{attribute 'linkalways'} 
{attribute 'no_explicit_call' := 'This FB is a CLASS and must be accessed using methods or properties'}
{attribute 'enable_dynamic_creation'}
FUNCTION_BLOCK Node_F_VN_DetectBlobsExp EXTENDS VisionNode
VAR
    ipSrcImage : _ITcVnImage;
    ipBlobContours : _ITcVnContainer;
    stParams : _TcVnParamsBlobDetection;
    aOffset : _TcVnPoint;
    hrPrev : _HRESULT(S_OK);
	hresult : _HRESULT(S_OK);
END_VAR

METHOD PUBLIC  Clone : I_Node
VAR
	pNode : POINTER TO Node_F_VN_DetectBlobsExp;
END_VAR
pNode := __NEW(Node_F_VN_DetectBlobsExp);
Clone := pNode^;
END_METHOD

METHOD FB_init : BOOL
VAR_INPUT
	bInitRetains : BOOL; // if TRUE, the retain variables are initialized (warm start / cold start)
	bInCopyCode : BOOL;  // if TRUE, the instance afterwards gets moved into the copy code (online change)
END_VAR
AddInput('ipSrcImage', ipSrcImage);
AddInput('stParams', stParams);
AddInput('aOffset', aOffset);
AddInput('hrPrev', hrPrev);
AddOutput('ipBlobContours', ipBlobContours);
AddOutput('hresult', hresult);
END_METHOD

METHOD PROTECTED OnExecute
hresult.Value := F_VN_DetectBlobsExp(
	ipSrcImage := ipSrcImage.Value,
    ipBlobContours := ipBlobContours.Value,
    stParams := stParams.Value,
    aOffset := aOffset.Value,
	hrPrev:= hrPrev.Value);
END_METHOD

METHOD PUBLIC PreExecutionCheck
VAR_INPUT
	Check : I_PreExecutionChecks;
END_VAR
Check.IsTrue(ipSrcImage.IsValid, 'ipSrcImage must contain an image');
Check.IsTrue((ipSrcImage.IsPixelDepth(8) OR ipSrcImage.IsPixelDepth(32)), 'ipSrcImage must be 8 or 32 bit pixel depth');
Check.IsTrue((ipSrcImage.HasChannelCount(1) OR ipSrcImage.HasChannelCount(3)), 'ipSrcImage must contain 1 or 3 channels');
Check.IsTrue(stParams.Value.fMaxThreshold >= stParams.Value.fMinThreshold, 'fMaxThreshold must be greater than or equal to fMinThreshold');
END_METHOD

END_FUNCTION_BLOCK

(* stored: Version 1.1.0.1, ProductVersion 3.1.4026.18
   POU Node_F_VN_DetectBlobsExp: Id {a7966657-125c-0d2b-32fa-81ffe10221c8}, SpecialFunc None
   Folder Constructor: Id {bbc10436-0102-05b7-2a51-3c32a270b36e}
   Method Clone: Id {25bd43b8-17ef-0404-3b99-a3d69c5d11e2}
   Method FB_init: Id {25aaaa77-b7d6-07c3-10e2-a0f8986286a8}
   Method OnExecute: Id {c8d94f75-57ef-00e1-2b84-2a416c29f207}
   Method PreExecutionCheck: Id {8c67a0a3-8e9f-0d85-3f77-6ba8f6e985d6} *)
